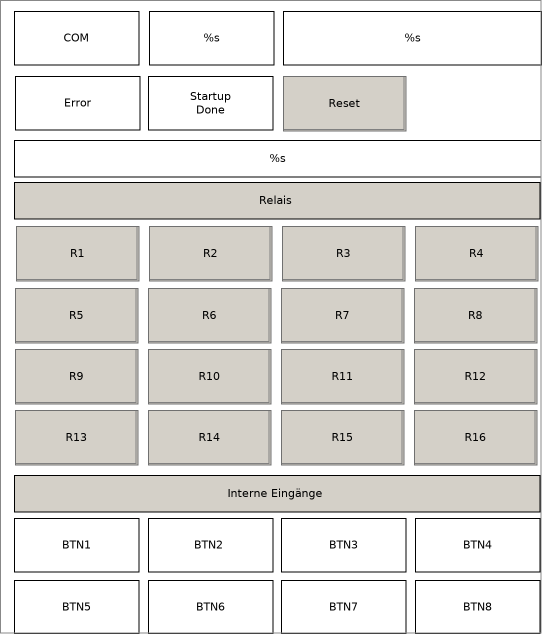
VISUALIZATION BusRelais16F_Frame  // 542x634
VAR_IN_OUT
	ST_BusRelais16F_Input		:ST_BusRelais16F_Input;
	ST_BusRelais16F_Output		:ST_BusRelais16F_Output;
	ST_BusRelais16F_Cnt			:ST_BusRelais16F_Cnt;
END_VAR
    Rectangle (14,11 125x54), "COM", colour toggle: ST_BusRelais16F_Output.bCOM
    Rectangle (14,518 125x54), "BTN1", colour toggle: ST_BusRelais16F_Output.bInputs[1]
    Rectangle (149,11 125x54), "%s", text variable: ST_BusRelais16F_Input.diID
    Rectangle (283,11 259x54), "%s", text variable: ST_BusRelais16F_Input.sName
    Rectangle (148,518 125x54), "BTN2", colour toggle: ST_BusRelais16F_Output.bInputs[2]
    Rectangle (281,518 125x54), "BTN3", colour toggle: ST_BusRelais16F_Output.bInputs[3]
    Rectangle (415,518 125x54), "BTN4", colour toggle: ST_BusRelais16F_Output.bInputs[4]
    Rectangle (14,580 125x54), "BTN5", colour toggle: ST_BusRelais16F_Output.bInputs[5]
    Rectangle (148,580 125x54), "BTN6", colour toggle: ST_BusRelais16F_Output.bInputs[6]
    Button (283,76 123x55), "Reset"
        tap ST_BusRelais16F_Input.bReset
    Rectangle (15,76 125x54), "Error", colour toggle: ST_BusRelais16F_Output.bError
    Rectangle (14,140 527x37), "%s", text variable: ST_BusRelais16F_Output.sState
    Rectangle (148,76 125x54), "Startup Done", colour toggle: ST_BusRelais16F_Output.bStartupDone
    Rectangle (14,475 526x37), "Interne Eingänge"
    Rectangle (281,580 125x54), "BTN7", colour toggle: ST_BusRelais16F_Output.bInputs[7]
    Rectangle (415,580 125x54), "BTN8", colour toggle: ST_BusRelais16F_Output.bInputs[8]
    Button (16,226 123x55), "R1"
        toggle ST_BusRelais16F_Input.bOut[1]
    Rectangle (14,182 526x37), "Relais"
    Button (149,226 123x55), "R2"
        toggle ST_BusRelais16F_Input.bOut[2]
    Button (282,226 123x55), "R3"
        toggle ST_BusRelais16F_Input.bOut[3]
    Button (415,226 123x55), "R4"
        toggle ST_BusRelais16F_Input.bOut[4]
    Button (15,288 123x55), "R5"
        toggle ST_BusRelais16F_Input.bOut[5]
    Button (148,288 123x55), "R6"
        toggle ST_BusRelais16F_Input.bOut[6]
    Button (281,288 123x55), "R7"
        toggle ST_BusRelais16F_Input.bOut[7]
    Button (414,288 123x55), "R8"
        toggle ST_BusRelais16F_Input.bOut[8]
    Button (15,349 123x55), "R9"
        toggle ST_BusRelais16F_Input.bOut[9]
    Button (148,349 123x55), "R10"
        toggle ST_BusRelais16F_Input.bOut[10]
    Button (281,349 123x55), "R11"
        toggle ST_BusRelais16F_Input.bOut[11]
    Button (414,349 123x55), "R12"
        toggle ST_BusRelais16F_Input.bOut[12]
    Button (15,410 123x55), "R13"
        toggle ST_BusRelais16F_Input.bOut[13]
    Button (148,410 123x55), "R14"
        toggle ST_BusRelais16F_Input.bOut[14]
    Button (281,410 123x55), "R15"
        toggle ST_BusRelais16F_Input.bOut[15]
    Button (414,410 123x55), "R16"
        toggle ST_BusRelais16F_Input.bOut[16]
END_VISUALIZATION

(* stored: Version 1.1.0.1, ProductVersion 3.1.4024.12
   Visu BusRelais16F_Frame: Id {f20b2591-9b36-4c16-b233-a47faa8baa12} *)
